FUNCTION_BLOCK EventWrapper_Produce_Green (* Composite Function Block Type *)
  (* Standard: 61499-2 *)
  (* Version 0.0, 4/9/2019, erik, nxtControl GmbH, template *)
  PACKAGE Main;
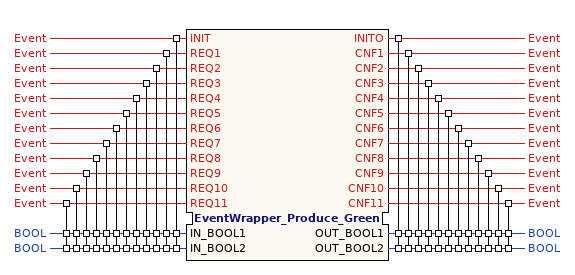
  EVENT_INPUT
    INIT WITH IN_BOOL1, IN_BOOL2; (* Initialization Request *)
    REQ1 WITH IN_BOOL1, IN_BOOL2; (* Normal Execution Request *)
    REQ2 WITH IN_BOOL1, IN_BOOL2;
    REQ3 WITH IN_BOOL1, IN_BOOL2;
    REQ4 WITH IN_BOOL1, IN_BOOL2;
    REQ5 WITH IN_BOOL1, IN_BOOL2;
    REQ6 WITH IN_BOOL1, IN_BOOL2;
    REQ7 WITH IN_BOOL1, IN_BOOL2;
    REQ8 WITH IN_BOOL1, IN_BOOL2;
    REQ9 WITH IN_BOOL1, IN_BOOL2;
    REQ10 WITH IN_BOOL1, IN_BOOL2;
    REQ11 WITH IN_BOOL1, IN_BOOL2;
  END_EVENT
  EVENT_OUTPUT
    INITO WITH OUT_BOOL1, OUT_BOOL2; (* Initialization Confirm *)
    CNF1 WITH OUT_BOOL1, OUT_BOOL2; (* Execution Confirmation *)
    CNF2 WITH OUT_BOOL1, OUT_BOOL2;
    CNF3 WITH OUT_BOOL1, OUT_BOOL2;
    CNF4 WITH OUT_BOOL1, OUT_BOOL2;
    CNF5 WITH OUT_BOOL1, OUT_BOOL2;
    CNF6 WITH OUT_BOOL1, OUT_BOOL2;
    CNF7 WITH OUT_BOOL1, OUT_BOOL2;
    CNF8 WITH OUT_BOOL1, OUT_BOOL2;
    CNF9 WITH OUT_BOOL1, OUT_BOOL2;
    CNF10 WITH OUT_BOOL1, OUT_BOOL2;
    CNF11 WITH OUT_BOOL1, OUT_BOOL2;
  END_EVENT
  VAR_INPUT
    IN_BOOL1 : BOOL;
    IN_BOOL2 : BOOL;
  END_VAR
  VAR_OUTPUT
    OUT_BOOL1 : BOOL;
    OUT_BOOL2 : BOOL;
  END_VAR
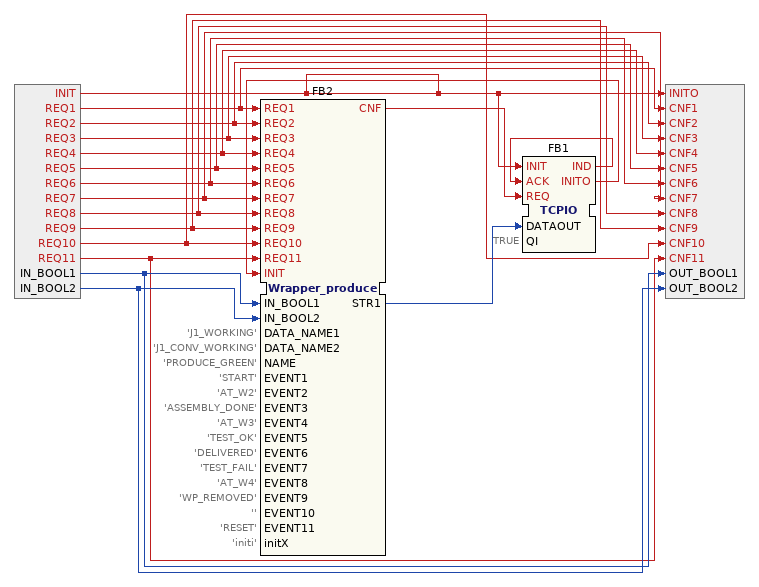
  FBS
    FB1 : TCPIO(QI := TRUE);
    FB2 : Wrapper_produce(DATA_NAME1 := 'J1_WORKING', DATA_NAME2 := 'J1_CONV_WORKING', NAME := 'PRODUCE_GREEN', EVENT1 := 'START', EVENT2 := 'AT_W2', EVENT3 := 'ASSEMBLY_DONE', EVENT4 := 'AT_W3', EVENT5 := 'TEST_OK', EVENT6 := 'DELIVERED', EVENT7 := 'TEST_FAIL', EVENT8 := 'AT_W4', EVENT9 := 'WP_REMOVED', EVENT10 := '', EVENT11 := 'RESET', initX := 'initi');
  END_FBS
  EVENT_CONNECTIONS
    INIT TO FB1.INIT;
    FB1.IND TO FB1.ACK;
    REQ1 TO FB2.REQ1;
    REQ2 TO FB2.REQ2;
    REQ3 TO FB2.REQ3;
    REQ4 TO FB2.REQ4;
    REQ5 TO FB2.REQ5;
    REQ6 TO FB2.REQ6;
    REQ7 TO FB2.REQ7;
    REQ8 TO FB2.REQ8;
    REQ9 TO FB2.REQ9;
    REQ10 TO FB2.REQ10;
    REQ11 TO FB2.REQ11;
    INIT TO INITO;
    REQ1 TO CNF1;
    REQ2 TO CNF2;
    REQ3 TO CNF3;
    REQ4 TO CNF4;
    REQ5 TO CNF5;
    REQ6 TO CNF6;
    REQ7 TO CNF7;
    REQ8 TO CNF8;
    REQ9 TO CNF9;
    REQ10 TO CNF10;
    REQ11 TO CNF11;
    FB1.INITO TO FB2.INIT;
    FB2.CNF TO FB1.REQ;
  END_CONNECTIONS
  DATA_CONNECTIONS
    IN_BOOL1 TO FB2.IN_BOOL1;
    IN_BOOL2 TO FB2.IN_BOOL2;
    IN_BOOL1 TO OUT_BOOL1;
    IN_BOOL2 TO OUT_BOOL2;
    FB2.STR1 TO FB1.DATAOUT;
  END_CONNECTIONS
END_FUNCTION_BLOCK
